{attribute addProperty BoxType "EL2889-0000-0016"}
{attribute addProperty Id "ChannelAT %Q*ARRAY[0..15] OF Channel_7F374EB0128160WcStateAT %I*WcState_28A8677510.1250InfoDataAT %I*InfoData_192954DE1620"}
{attribute addProperty CRC "924279498"}
{attribute addProperty SizeInBites "145"}
{attribute addProperty SizeInBytes "18.125"}
TYPE EL2889_859F43D2 :
STRUCT
	{attribute addProperty Name "Channel"}
	Channel : ARRAY[0..15] OF Channel_7F374EB0;
	{attribute addProperty Name "WcState"}
	WcState : WcState_28A86775;
	{attribute addProperty Name "InfoData"}
	InfoData : InfoData_192954DE;
END_STRUCT
END_TYPE

(* stored: Version 1.2.0.0, ProductVersion 3.1.4024.9
   DUT EL2889_859F43D2: Id {41690d6b-42af-42d9-94a9-6218e49af1f1} *)
